FUNCTION_BLOCK F_ROUND (* Service Interface Function Block Type *)
  (* Standard: 61499-2 *)
  (* Version 0.0, 2011-07-21, 4DIAC-IDE, 4DIAC-Consortium *)
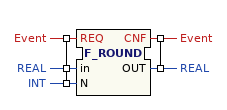
  EVENT_INPUT
    REQ WITH in, N; (* Service Request *)
  END_EVENT
  EVENT_OUTPUT
    CNF WITH OUT; (* Confirmation of Requested Service *)
  END_EVENT
  VAR_INPUT
    in : REAL; (* Input for round *)
    N : INT; (* Digits behind comma *)
  END_VAR
  VAR_OUTPUT
    OUT : REAL; (* Round outcome *)
  END_VAR
END_FUNCTION_BLOCK
